// TIA Portal V16 export
// export: Created 2025-08-01T13:38:14.8015943Z, ExportSetting WithDefaults, DisplayName Totally Integrated Automation Portal, DisplayVersion V16, DisplayName TIA Portal Version Control Interface, DisplayVersion V16, DisplayName TIA Portal Openness, DisplayVersion V16, DisplayName STEP 7 Professional, DisplayVersion V16, DisplayName STEP 7 Safety, DisplayVersion V16, DisplayName WinCC Advanced, DisplayVersion V16
VAR_GLOBAL   // PLC tag table "PositionControl"
   Counter1_IW100 AT %IW100 : Int;
   Counter2_IW102 AT %IW102 : Int;
   "Manual Jog Fwd" AT %M137.0 : Bool;
   "Manual Jog Rev" AT %M137.1 : Bool;
   ReferenceSwitchAxis3 AT %I3.0 : Bool;
   EncoderBand_Alive AT %IW110 : Int;
   EncoderBand_RawCounter AT %ID112 : DInt;
   EncoderBand_FineCounter AT %IW113 : Int;
   Zpuls_Encoder_Band AT %I110.3 : Bool;
   Enc1 AT %ID110 : DInt;
   Enc2 AT %ID111 : DInt;
   Enc3 AT %ID113 : DInt;
   "Zpuls_Encoder_Band(1)" AT %I113.3 : Bool;
   "Enc3(1)" AT %ID114 : DInt;
   "Enc3(2)" AT %ID115 : DInt;
   "Enc3(3)" AT %ID116 : DInt;
   "Enc3(4)" AT %ID117 : DInt;
   "Enc3(5)" AT %ID118 : DInt;
   "Enc3(6)" AT %IW112 : Int;
   Enable AT %QW110 : Word;
   MovePos2 AT %M222.0 : Bool;
   ActivateProductBufferV3 AT %M222.1 : Bool;
END_VAR
